// TwinCAT 3 PLC project PLC
// ProgramVersion: 3.1.4026.19
// CompilerDefines: VISU_USEPROPERTYINFO
// libraries:
//   Tc2_Standard, * (Beckhoff Automation GmbH)
//   Tc2_System, * (Beckhoff Automation GmbH)
//   VisuDialogs, * (System)
// project tree:
//   / GlobalTextList.TcGTLO, PlcTask.TcTTO, Visualization Manager.TcVMO (not stored)
//   POUs/ MAIN.TcPOU
//   VISUs/ Visualization.TcVIS
// real-time tasks:
//   TASK PlcTask: cycle T#10ms, priority 20, ADS port 350

CONFIGURATION PLC
    RESOURCE PLC ON TwinCAT3
        TASK PlcTask(INTERVAL := T#10ms, PRIORITY := 20);
        PROGRAM MAIN WITH PlcTask : MAIN;
    END_RESOURCE
END_CONFIGURATION

// ---- POUs/MAIN.TcPOU
PROGRAM MAIN
VAR
	fActualValue : REAL;
	fTargetValue : REAL := 50.0 ;
	fTolerance : REAL := 2.0 ;
	
	bTargetReached : BOOL;
END_VAR

IF (fActualValue >= (fTargetValue - fTolerance)) AND (FaCTUALvALUE <= (fTargetValue + fTolerance)) THEN
	bTargetReached := TRUE;
ELSE
	bTargetReached := FALSE;
END_IF

END_PROGRAM

// ---- GlobalTextList.TcGTLO
TEXTLIST GlobalTextList
  343 = 'Ziel: %.1f'
  425 = 'Ziel: %.f'
END_TEXTLIST

// ---- VISUs/Visualization.TcVIS
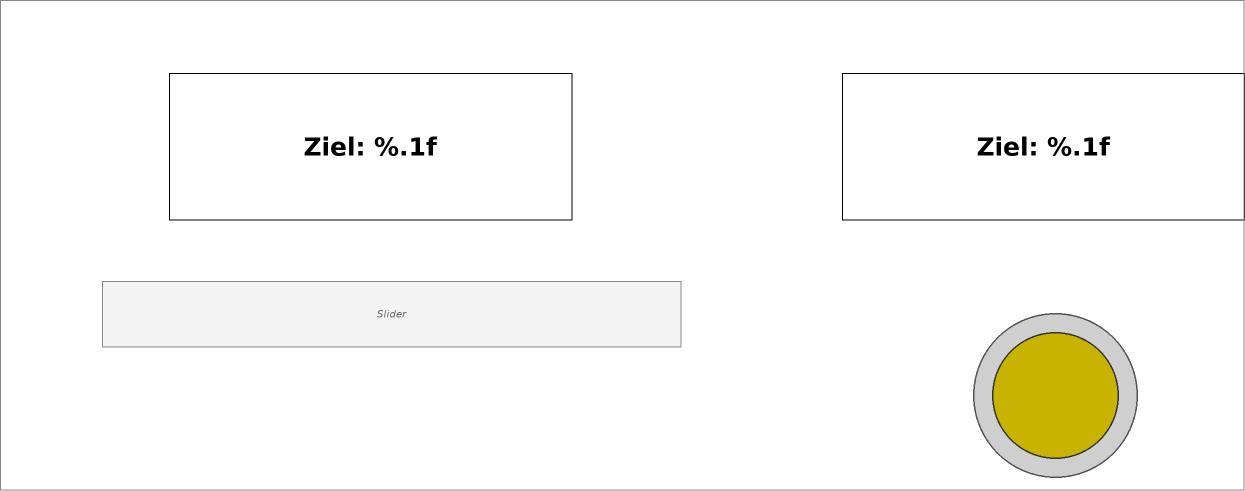
VISUALIZATION Visualization  // 1245x491
    Rectangle (842,73 403x147), "Ziel: %.1f", text variable: MAIN.fTargetValue
        OnMouseClick: write MAIN.fTargetValue via VisuDialogs.Numpad
    Slider (102,281 579x66), variable: MAIN.fActualValue, scale 0..100
    Rectangle (169,73 403x147), "Ziel: %.1f", text variable: MAIN.fActualValue
        OnMouseClick: write MAIN.fTargetValue via VisuDialogs.Numpad
    Lamp1 (956,300 199x191), variable: MAIN.bTargetReached, style: Lamp-Lamp1-Yellow
END_VISUALIZATION
